FUNCTION_BLOCK CM_SensorAnalog_V2
VAR_INPUT
	
	PI_ManualMode : BOOL;
	PI_AutoMode : BOOL;
	
	//ALARMS:
	PI_AlarmHighHighEnable : BOOL;
	PI_AlarmHighEnable : BOOL;
	PI_AlarmLowEnable : BOOL;
	PI_AlarmLowLowEnable : BOOL;
	
	PI_AlarmHighHighLimit : REAL;
	PI_AlarmHighLimit : REAL;
	PI_AlarmLowLimit : REAL;
	PI_AlarmLowLowLimit : REAL;
	
	PI_AlarmDelay_HH : LREAL;
	PI_AlarmDelay_H : LREAL;
	PI_AlarmDelay_L : LREAL;
	PI_AlarmDelay_LL : LREAL;
	
	PI_PV :DINT;
	
	
	ENABLE_SCALING : BOOL;
	PI_PV_MAX_IN : INT;
	PI_PV_MIN_IN : INT;
	PI_PV_MAX_OUT : INT;
	PI_PV_MIN_OUT : INT;
END_VAR
VAR_OUTPUT
	
	PO_PV_SCALED : REAL;

	PO_ALARM_HH : BOOL;
	PO_ALARM_H : BOOL;
	PO_ALARM_L : BOOL;
	PO_ALARM_LL : BOOL;
END_VAR
VAR
	scale : Tc2_ControllerToolbox.FB_CTRL_SCALE;
	scaleParams : ST_CTRL_SCALE_PARAMS;
	
	Alarm_limit_Exceeded_HH : BOOL;
	Alarm_limit_Exceeded_H : BOOL;
	Alarm_limit_Exceeded_L : BOOL;
	Alarm_limit_Exceeded_LL : BOOL;
	
	Alarm_Ack_HH : BOOL;
	Alarm_Ack_H : BOOL;
	Alarm_Ack_L : BOOL;
	Alarm_Ack_LL : BOOL;
	
	alarmDelay_HH : systemTimeDelay;
	alarmDelay_H : systemTimeDelay;
	alarmDelay_L : systemTimeDelay;
	alarmDelay_LL : systemTimeDelay;
	
	DelayForHistorianBit_HH: TON;
	DelayForHistorianBit_H: TON;
	DelayForHistorianBit_L: TON;
	DelayForHistorianBit_LL: TON;
	
	HIST_BIT_HH : BOOL;
	HIST_BIT_H : BOOL;
	HIST_BIT_L : BOOL;
	HIST_BIT_LL : BOOL;
END_VAR
VAR_IN_OUT
END_VAR

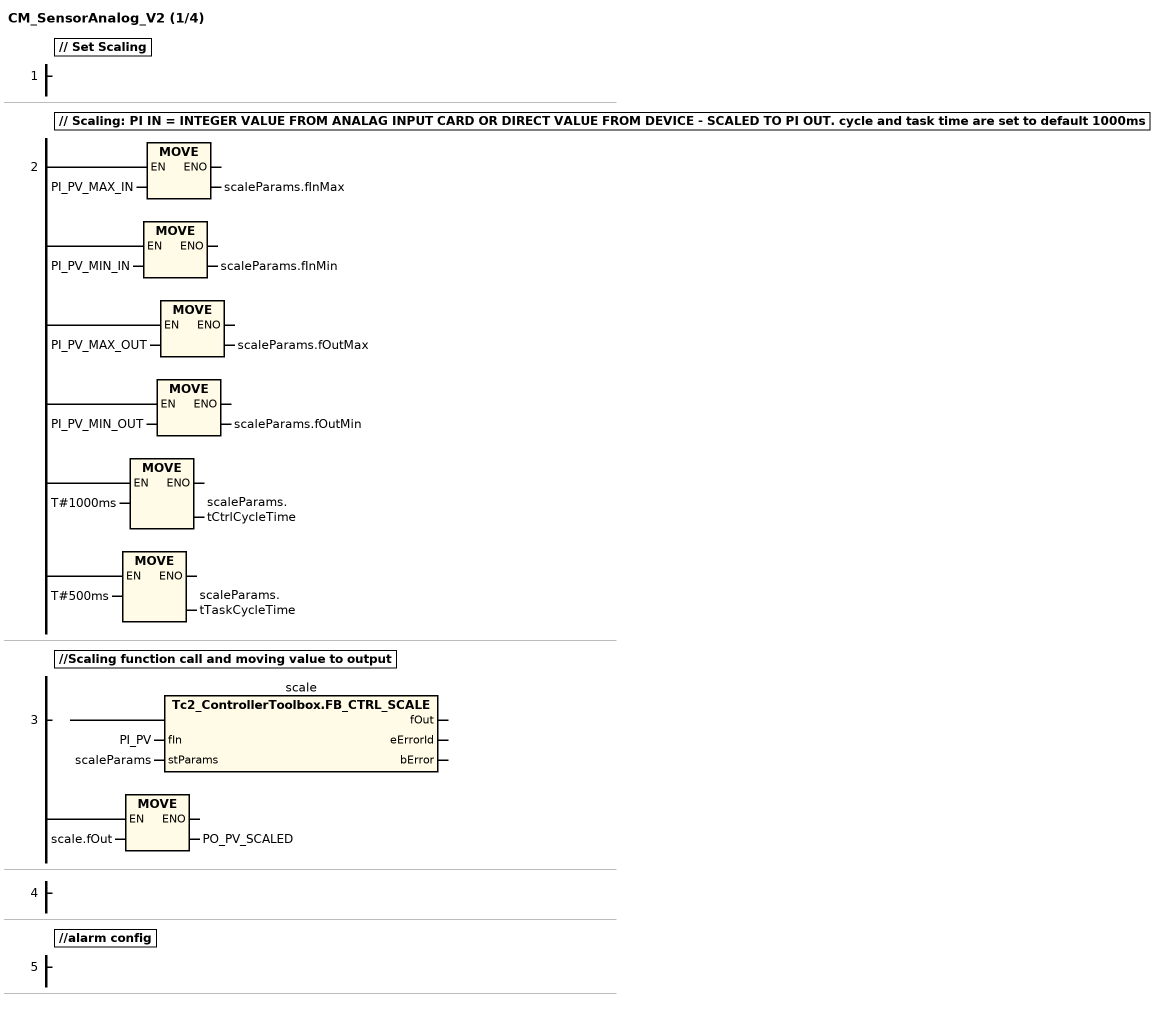
// NETWORK 1
// label: // Set Scaling

// NETWORK 2
// label: // Scaling: PI IN = INTEGER VALUE FROM ANALAG INPUT CARD OR DIRECT VALUE FROM DEVICE - SCALED TO PI OUT. cycle and task time are set to default 1000ms
scaleParams.fInMax := PI_PV_MAX_IN;
scaleParams.fInMin := PI_PV_MIN_IN;
scaleParams.fOutMax := PI_PV_MAX_OUT;
scaleParams.fOutMin := PI_PV_MIN_OUT;
scaleParams.tCtrlCycleTime := T#1000ms;
scaleParams.tTaskCycleTime := T#500ms;

// NETWORK 3
// label: //Scaling function call and moving value to output
scale(fIn := PI_PV, stParams := scaleParams); // Tc2_ControllerToolbox.FB_CTRL_SCALE
PO_PV_SCALED := scale.fOut;

// NETWORK 4

// NETWORK 5
// label: //alarm config

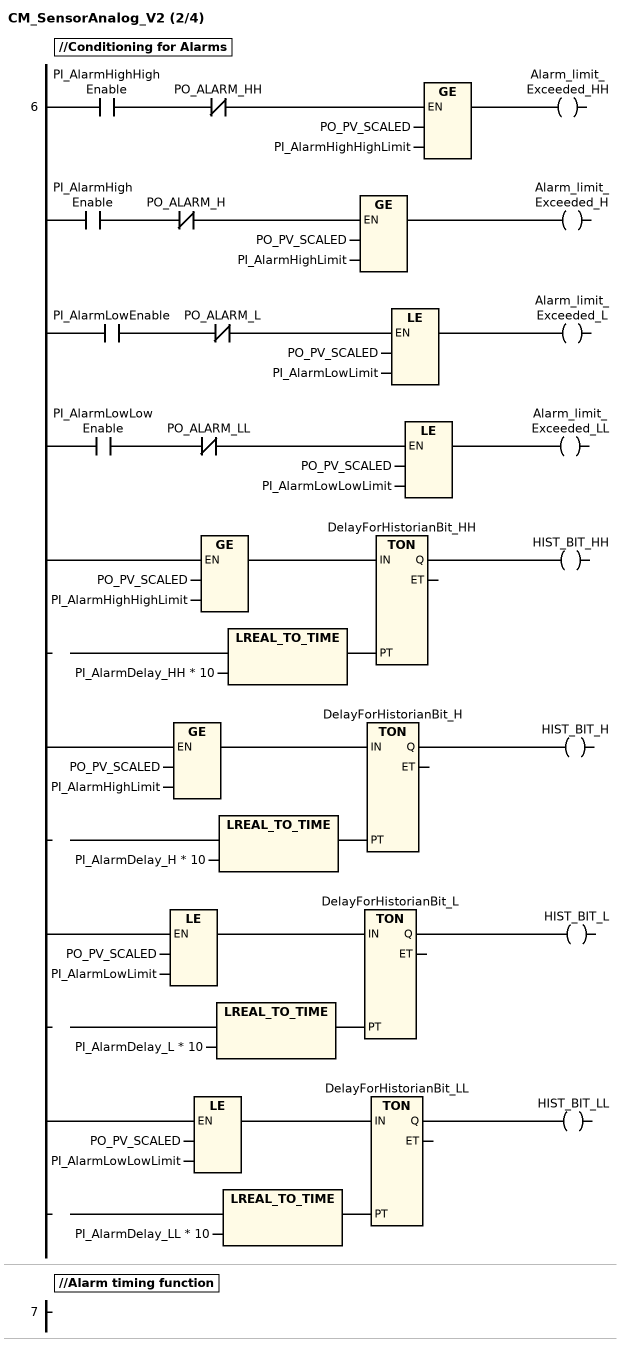
// NETWORK 6
// label: //Conditioning for Alarms
Alarm_limit_Exceeded_HH := PI_AlarmHighHighEnable AND NOT PO_ALARM_HH AND PO_PV_SCALED >= PI_AlarmHighHighLimit;
Alarm_limit_Exceeded_H := PI_AlarmHighEnable AND NOT PO_ALARM_H AND PO_PV_SCALED >= PI_AlarmHighLimit;
Alarm_limit_Exceeded_L := PI_AlarmLowEnable AND NOT PO_ALARM_L AND PO_PV_SCALED <= PI_AlarmLowLimit;
Alarm_limit_Exceeded_LL := PI_AlarmLowLowEnable AND NOT PO_ALARM_LL AND PO_PV_SCALED <= PI_AlarmLowLowLimit;
DelayForHistorianBit_HH(IN := PO_PV_SCALED >= PI_AlarmHighHighLimit, PT := LREAL_TO_TIME(PI_AlarmDelay_HH * 10)); // TON
HIST_BIT_HH := DelayForHistorianBit_HH.Q;
DelayForHistorianBit_H(IN := PO_PV_SCALED >= PI_AlarmHighLimit, PT := LREAL_TO_TIME(PI_AlarmDelay_H * 10)); // TON
HIST_BIT_H := DelayForHistorianBit_H.Q;
DelayForHistorianBit_L(IN := PO_PV_SCALED <= PI_AlarmLowLimit, PT := LREAL_TO_TIME(PI_AlarmDelay_L * 10)); // TON
HIST_BIT_L := DelayForHistorianBit_L.Q;
DelayForHistorianBit_LL(IN := PO_PV_SCALED <= PI_AlarmLowLowLimit, PT := LREAL_TO_TIME(PI_AlarmDelay_LL * 10)); // TON
HIST_BIT_LL := DelayForHistorianBit_LL.Q;

// NETWORK 7
// label: //Alarm timing function

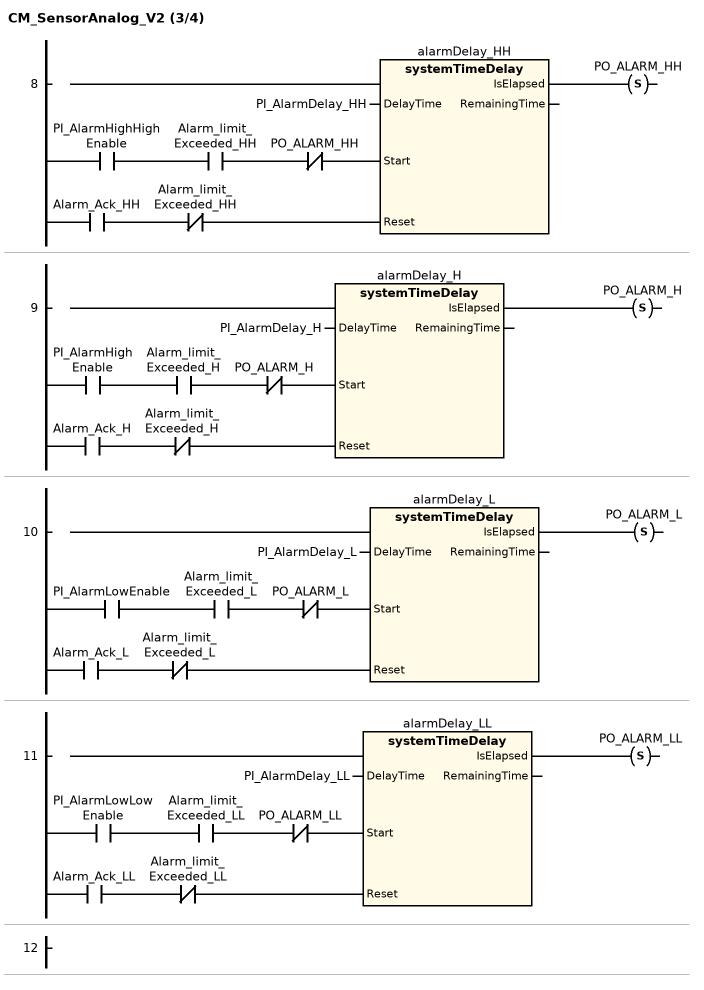
// NETWORK 8
alarmDelay_HH(
    DelayTime := PI_AlarmDelay_HH,
    Start := PI_AlarmHighHighEnable AND Alarm_limit_Exceeded_HH AND NOT PO_ALARM_HH,
    Reset := Alarm_Ack_HH AND NOT Alarm_limit_Exceeded_HH); // systemTimeDelay
PO_ALARM_HH S= alarmDelay_HH.IsElapsed;

// NETWORK 9
alarmDelay_H(
    DelayTime := PI_AlarmDelay_H,
    Start := PI_AlarmHighEnable AND Alarm_limit_Exceeded_H AND NOT PO_ALARM_H,
    Reset := Alarm_Ack_H AND NOT Alarm_limit_Exceeded_H); // systemTimeDelay
PO_ALARM_H S= alarmDelay_H.IsElapsed;

// NETWORK 10
alarmDelay_L(
    DelayTime := PI_AlarmDelay_L,
    Start := PI_AlarmLowEnable AND Alarm_limit_Exceeded_L AND NOT PO_ALARM_L,
    Reset := Alarm_Ack_L AND NOT Alarm_limit_Exceeded_L); // systemTimeDelay
PO_ALARM_L S= alarmDelay_L.IsElapsed;

// NETWORK 11
alarmDelay_LL(
    DelayTime := PI_AlarmDelay_LL,
    Start := PI_AlarmLowLowEnable AND Alarm_limit_Exceeded_LL AND NOT PO_ALARM_LL,
    Reset := Alarm_Ack_LL AND NOT Alarm_limit_Exceeded_LL); // systemTimeDelay
PO_ALARM_LL S= alarmDelay_LL.IsElapsed;

// NETWORK 12

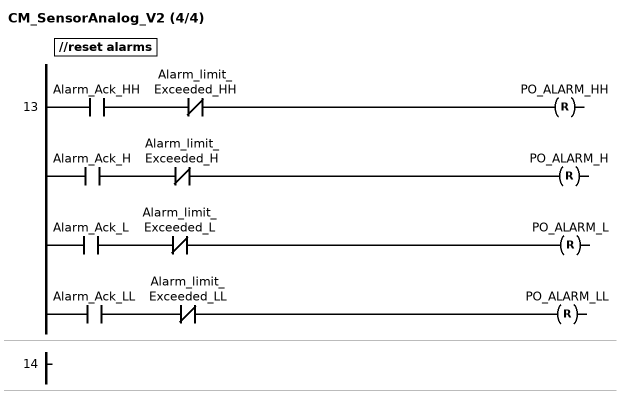
// NETWORK 13
// label: //reset alarms
PO_ALARM_HH R= Alarm_Ack_HH AND NOT Alarm_limit_Exceeded_HH;
PO_ALARM_H R= Alarm_Ack_H AND NOT Alarm_limit_Exceeded_H;
PO_ALARM_L R= Alarm_Ack_L AND NOT Alarm_limit_Exceeded_L;
PO_ALARM_LL R= Alarm_Ack_LL AND NOT Alarm_limit_Exceeded_LL;

// NETWORK 14

END_FUNCTION_BLOCK

(* stored: Version 1.1.0.1, ProductVersion 3.1.4024.13
   POU CM_SensorAnalog_V2: Id {4a9e58f3-a0b0-49a4-8a8b-f0da4bcd6505}, SpecialFunc None *)
